(* CODESYS project hmi_library.library
   Author: AMKO-Engineering
   Placeholder: HMI_Library
   Title: HMI_Library
   Version: 1.0.0.3
   Description: Basic HMI screens for use with Utilities and device libraries
   Company: AMKO-Engineering

Project tree, tasks and I/O mapping:
  libraries: CmpBitmapPool, 3.5.7.0 (System); Device_Library, 1.2.0.3 (AMKO-Engineering); System_Library, * (AMKO-Engineering); Utilities_Library, 1.2.0.3 (AMKO-Engineering); VisuDialogs, 3.5.12.0 (System)
  BaseScreens/
  GVL/
    data type E_StartVisu
    global variables GVL_HMI
  IconsAndPictures/
    Backgrounds/
      Background.svg
      Background_Bottom.svg
      Background_Bottomzonder knop.png
      Background_Sides.svg
      image pool BackgroundImagePool
      Emergency Stop Active.jpg
    Buttons/
      Home Button/
        Home Settings switch.png
        Home_Settings switch.svg
        Home-Settings Switch Pushed.png
        Home-Settings Switch Pushed.svg
      Screen Buttons/
        Power Off Pressed.png
        Power off.png
        To Parameter Screen Pressed.png
        To Parameter Screen Pressed.svg
        To Parameter Screen.png
        To Parameter Screen.svg
      image pool ButtonImagePool
    Logos/
      Amko Basis.svg
      Logo Dark blue.svg
      image pool LogoPool
  00000000-0000-0000-0000-000000000000|IconsAndPictures\Backgrounds\Background.svg
  00000000-0000-0000-0000-000000000000|IconsAndPictures\Backgrounds\Background_Bottom.svg
  00000000-0000-0000-0000-000000000000|IconsAndPictures\Backgrounds\Background_Bottomzonder knop.png
  00000000-0000-0000-0000-000000000000|IconsAndPictures\Backgrounds\Background_Sides.svg
  00000000-0000-0000-0000-000000000000|IconsAndPictures\Backgrounds\Emergency Stop Active.jpg
  00000000-0000-0000-0000-000000000000|IconsAndPictures\Buttons\Home Button\Home Settings switch.png
  00000000-0000-0000-0000-000000000000|IconsAndPictures\Buttons\Home Button\Home_Settings switch.svg
  00000000-0000-0000-0000-000000000000|IconsAndPictures\Buttons\Home Button\Home-Settings Switch Pushed.png
  00000000-0000-0000-0000-000000000000|IconsAndPictures\Buttons\Home Button\Home-Settings Switch Pushed.svg
  00000000-0000-0000-0000-000000000000|IconsAndPictures\Buttons\Screen Buttons\Power Off Pressed.png
  00000000-0000-0000-0000-000000000000|IconsAndPictures\Buttons\Screen Buttons\Power off.png
  00000000-0000-0000-0000-000000000000|IconsAndPictures\Buttons\Screen Buttons\To Parameter Screen Pressed.png
  00000000-0000-0000-0000-000000000000|IconsAndPictures\Buttons\Screen Buttons\To Parameter Screen Pressed.svg
  00000000-0000-0000-0000-000000000000|IconsAndPictures\Buttons\Screen Buttons\To Parameter Screen.png
  00000000-0000-0000-0000-000000000000|IconsAndPictures\Buttons\Screen Buttons\To Parameter Screen.svg
  00000000-0000-0000-0000-000000000000|IconsAndPictures\Logos\Amko Basis.svg
  00000000-0000-0000-0000-000000000000|IconsAndPictures\Logos\Logo Dark blue.svg
  InputFunctions/
    function block FB_HMIInputBase [ST]: SetHMIInstructions, SetOutputToPLC
    function block FB_HMILREALInput [ST]: SetOutputToPLC
  Screens/
    Backgrounds/
      visualisation BackgroundNoButton
    EventsAndMessage/
      visualisation BasicMessageScreen
      visualisation EstopScreen
    Manual/
      DeviceScreens/
        visualisation VisuAnalogOutControl
        visualisation VisuAnlogInputControl
        visualisation VisuAxisControl
        visualisation VisuCylinderControl
        visualisation VisuDigitalInputControl
        visualisation VisuDigitalOutControl
        visualisation VisuPushbuttonLightControl
        visualisation VisuPWMControl
        visualisation VisuUndefinedControl
        visualisation VisuValveControl
      visualisation ManualControl
    Parameter/
      visualisation ParameterScreen
    Startup Screen/
      visualisation LogoScreen
      visualisation StartScreen
  TextLists/
    text list E_ComponentTypes
    text list E_FaultTypes
    text list E_Locations
    text list E_MessageNumbers
    text list E_ParameterNames
    text list GlobalTextList
    text list TL_MessageDiscriptions
*)

// GVL/E_StartVisu
{attribute 'qualified_only'}
{attribute 'strict'}
TYPE E_StartVisu :
(
	Logo := 0,
	Parameter,
	Manual
);
END_TYPE

// GVL/GVL_HMI
{attribute 'qualified_only'}
VAR_GLOBAL
	nStartVisu	: E_StartVisu := E_StartVisu.Logo ;
END_VAR

// InputFunctions/FB_HMIInputBase
FUNCTION_BLOCK ABSTRACT FB_HMIInputBase //Base function for HMI inputs
VAR_INPUT
	bEnable : BOOL := TRUE ;
END_VAR
VAR_OUTPUT
	bInVisible			: BOOL := TRUE ; // input is visible (standard := NOT bEnable )
	bDeactivateInput	: BOOL := TRUE ; // input is enabled (Standard := bEnable)
END_VAR
VAR
END_VAR

SetHMIInstructions();

METHOD INTERNAL SetHMIInstructions : BOOL
VAR_INPUT
END_VAR
bInVisible 			:= NOT bEnable ;
bDeactivateInput	:= NOT bEnable ;
END_METHOD

METHOD ABSTRACT SetOutputToPLC : BOOL
VAR_INPUT
END_VAR
END_METHOD

END_FUNCTION_BLOCK

// InputFunctions/FB_HMILREALInput
FUNCTION_BLOCK PUBLIC FB_HMILREALInput EXTENDS FB_HMIInputBase // Analog value input from HMI
VAR_INPUT
	fInputFromHMI	: LREAL ;
END_VAR
VAR_OUTPUT
	fOutputToPLC	: LREAL ;
END_VAR
VAR
END_VAR

// call base function 
SUPER^();

// Set output to PLC
SetOutputToPLC();

METHOD PUBLIC SetOutputToPLC : BOOL
VAR_INPUT
END_VAR
IF bEnable THEN 
	fOutputToPLC := fInputFromHMI ;
END_IF
END_METHOD

END_FUNCTION_BLOCK

// Screens/Backgrounds/BackgroundNoButton
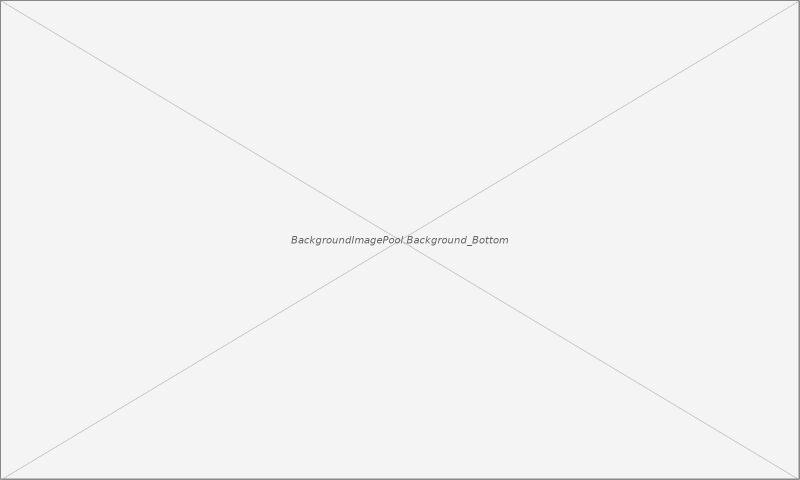
VISUALIZATION BackgroundNoButton  // 800x480
    Image (0,0 800x480), invisible if: SystemBase.bSystemOK, input disabled if: SystemBase.bSystemOK, image: BackgroundImagePool.Emergency Stop Active
    Image (0,0 800x480), image: BackgroundImagePool.Background_Bottom
END_VISUALIZATION

// Screens/EventsAndMessage/BasicMessageScreen
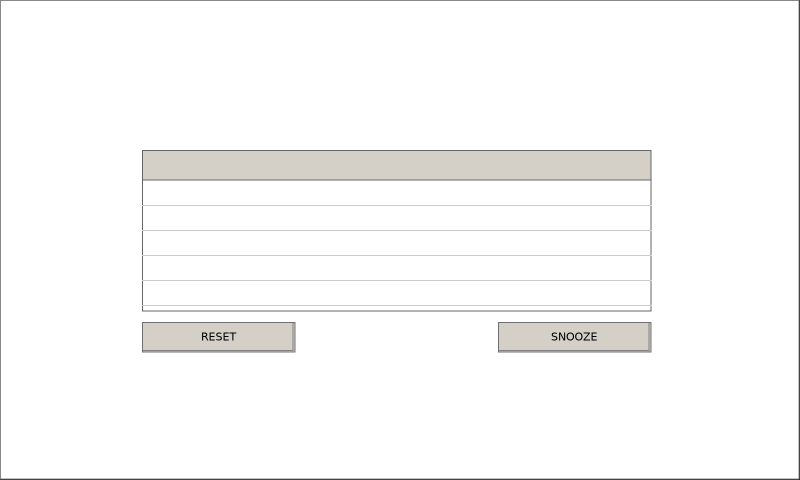
VISUALIZATION BasicMessageScreen  // 800x480
    Rectangle (0,0 800x480)
    Table (142,150 509x161), data array: Utilities_Library.GVL_Message.arActiveFaults
        p3854506369: Utilities_Library.GVL_Message.arActiveFaults[INDEX].Active
        p1892666644: Utilities_Library.GVL_Message.arActiveFaults[INDEX].FaultType
        p338671338: Utilities_Library.GVL_Message.arActiveFaults[INDEX].MessageNumber
        p2170511999: Utilities_Library.GVL_Message.arActiveFaults[INDEX].LocationNumber
        p3723444502: Utilities_Library.GVL_Message.arActiveFaults[INDEX].Discription
        p1218418051: Utilities_Library.GVL_Message.arActiveFaults[INDEX].LocationName
        p746581629: Utilities_Library.GVL_Message.arActiveFaults[INDEX].ComponentType
        p3104783080: Utilities_Library.GVL_Message.arActiveFaults[INDEX].StartTime
        p2501879983: Utilities_Library.GVL_Message.arActiveFaults[INDEX].EndTime
        p7306298: Utilities_Library.GVL_Message.arActiveFaults[INDEX].nModuleID
        p1933151965: Utilities_Library.GVL_Message.arActiveFaults[INDEX].FullFaultId
    Button (142,322 153x30), "RESET"
        tap Utilities_Library.GVL_Message.bResetFaults
    Button (498,322 153x30), "SNOOZE"
        tap Utilities_Library.GVL_Message.bCmdSnoozeMessage
END_VISUALIZATION

// Screens/EventsAndMessage/EstopScreen
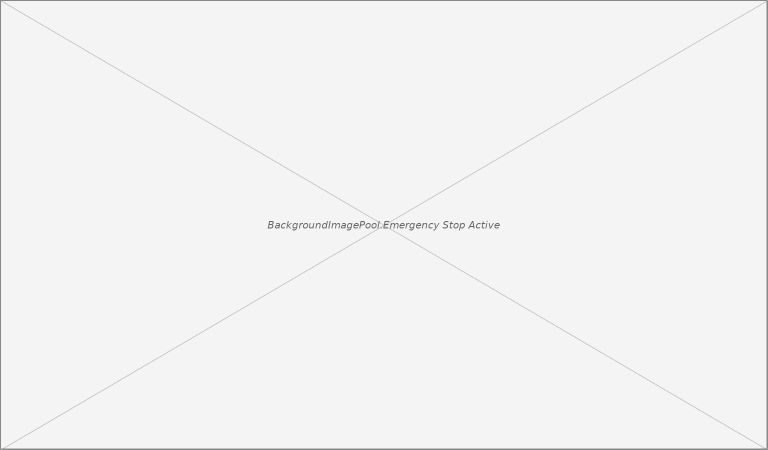
VISUALIZATION EstopScreen  // 768x450
    Image (0,0 768x450), image: BackgroundImagePool.Emergency Stop Active
END_VISUALIZATION

// Screens/Manual/DeviceScreens/VisuAnalogOutControl
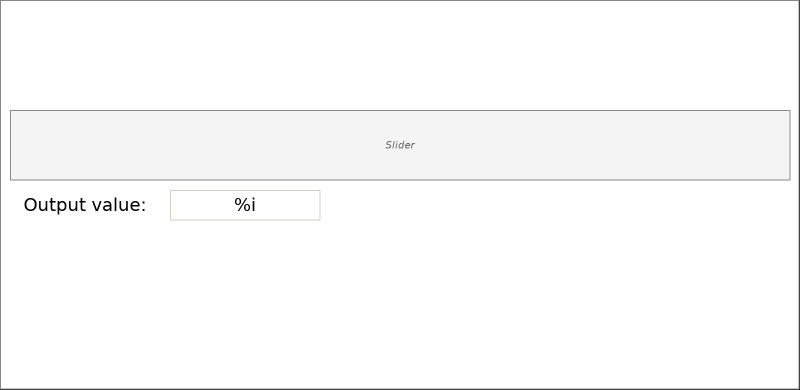
VISUALIZATION VisuAnalogOutControl  // 800x390
    Rectangle (0,0 800x390)
    Slider (10,110 780x70), variable: GVL_DevManual.fbManualControler.pDevAnalogOut^.fCmdValue, scale 0..100
    Textfield (170,190 150x30), "%i", text variable: GVL_DevManual.fbManualControler.pDevAnalogOut^.fCmdValue
        OnMouseClick: write the text variable via VisuDialogs.Numpad
    Label (10,190 150x30), "Output value:"
END_VISUALIZATION

// Screens/Manual/DeviceScreens/VisuAnlogInputControl
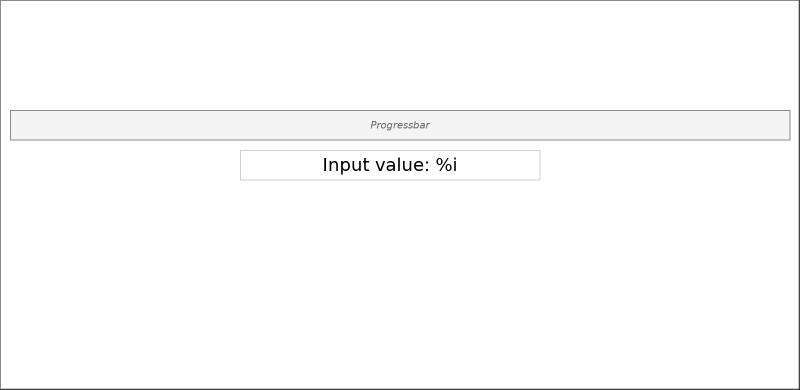
VISUALIZATION VisuAnlogInputControl  // 800x390
    Rectangle (0,0 800x390)
    Progressbar (10,110 780x30), variable: GVL_DevManual.fbManualControler.pDevAnalogInput^.fValue
    Textfield (240,150 300x30), "Input value: %i", text variable: GVL_DevManual.fbManualControler.pDevAnalogInput^.fValue
END_VISUALIZATION

// Screens/Manual/DeviceScreens/VisuAxisControl
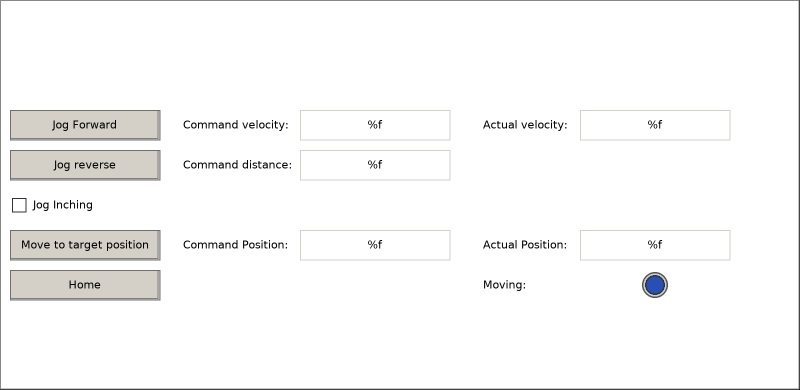
VISUALIZATION VisuAxisControl  // 800x390
    Rectangle (0,0 800x390)
    Button (10,110 150x30), "Jog Forward"
        tap GVL_DevManual.fbManualControler.pDevAxis^.stManualCtrl.bCmdJogForward
    Button (10,150 150x30), "Jog reverse"
        tap GVL_DevManual.fbManualControler.pDevAxis^.stManualCtrl.bCmdJogReverse
    Button (10,230 150x30), "Move to target position"
        tap GVL_DevManual.fbManualControler.pDevAxis^.stManualCtrl.bCmdToPos
    Button (10,270 150x30), "Home"
        tap GVL_DevManual.fbManualControler.pDevAxis^.stManualCtrl.bCmdHome
    Checkbox (10,190 150x30), "Jog Inching", variable: GVL_DevManual.fbManualControler.pDevAxis^.stManualCtrl.bCmdInching
    Label (180,150 120x30), "Command distance:"
    Label (180,110 120x30), "Command velocity:"
    Label (180,230 120x30), "Command Position:"
    Textfield (300,110 150x30), "%f", text variable: GVL_DevManual.fbManualControler.pDevAxis^.stManualCtrl.fVelocity
        OnMouseDown: write the text variable via VisuDialogs.Numpad
    Textfield (300,150 150x30), "%f", text variable: GVL_DevManual.fbManualControler.pDevAxis^.stManualCtrl.fDistance
        OnMouseDown: write the text variable via VisuDialogs.Numpad
    Textfield (300,230 150x30), "%f", text variable: GVL_DevManual.fbManualControler.pDevAxis^.stManualCtrl.fPosition
        OnMouseDown: write the text variable via VisuDialogs.Numpad
    Label (480,110 100x30), "Actual velocity:"
    Label (480,230 100x30), "Actual Position:"
    Textfield (580,230 150x30), "%f", text variable: GVL_DevManual.fbManualControler.pDevAxis^.fActPosition
        OnMouseDown: write the text variable via VisuDialogs.Numpad
    Textfield (580,110 150x30), "%f", text variable: GVL_DevManual.fbManualControler.pDevAxis^.fVelocity
        OnMouseDown: write the text variable via VisuDialogs.Numpad
    Lamp1 (580,270 150x30), variable: GVL_DevManual.fbManualControler.pDevAxis^.AxisRef.Status.Moving, style: Lamp-Lamp1-Blue
    Label (480,270 100x30), "Moving:"
END_VISUALIZATION

// Screens/Manual/DeviceScreens/VisuCylinderControl
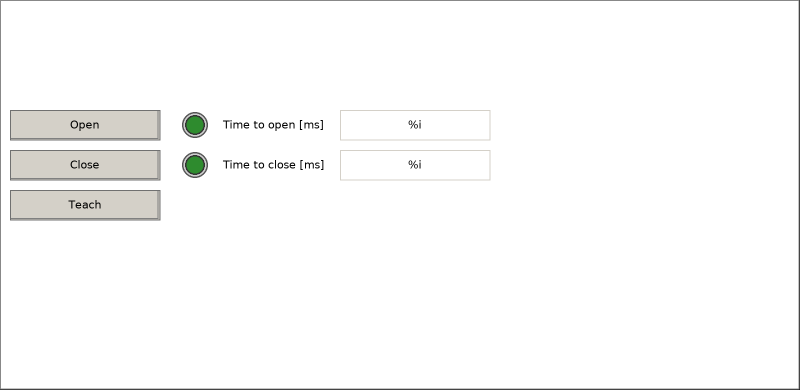
VISUALIZATION VisuCylinderControl  // 800x390
    Rectangle (0,0 800x390)
    Button (10,110 150x30), "Open"
        tap GVL_DevManual.fbManualControler.pDevCylinder^.stManualCtrl.bCmdOpen
    Button (10,150 150x30), "Close"
        tap GVL_DevManual.fbManualControler.pDevCylinder^.stManualCtrl.bCmdClose
    Lamp1 (180,110 30x30), variable: GVL_DevManual.fbManualControler.pDevCylinder^.bFco_Open, style: Lamp-Lamp1-Green
    Button (10,190 150x30), "Teach"
        toggle GVL_DevManual.fbManualControler.pDevCylinder^.stManualCtrl.bCmdTeach
    Lamp1 (180,150 30x30), variable: GVL_DevManual.fbManualControler.pDevCylinder^.bFco_Closed, style: Lamp-Lamp1-Green
    Label (220,110 100x30), "Time to open [ms]"
    Label (220,150 100x30), "Time to close [ms]"
    Textfield (340,150 150x30), "%i", text variable: GVL_DevManual.fbManualControler.pDevCylinder^.stParTimeToClose.fValue
        OnMouseClick: write the text variable via VisuDialogs.Numpad, min 0
    Textfield (340,110 150x30), "%i", text variable: GVL_DevManual.fbManualControler.pDevCylinder^.stParTimeToOpen.fValue
        OnMouseClick: write the text variable via VisuDialogs.Numpad, min 0
END_VISUALIZATION

// Screens/Manual/DeviceScreens/VisuDigitalInputControl
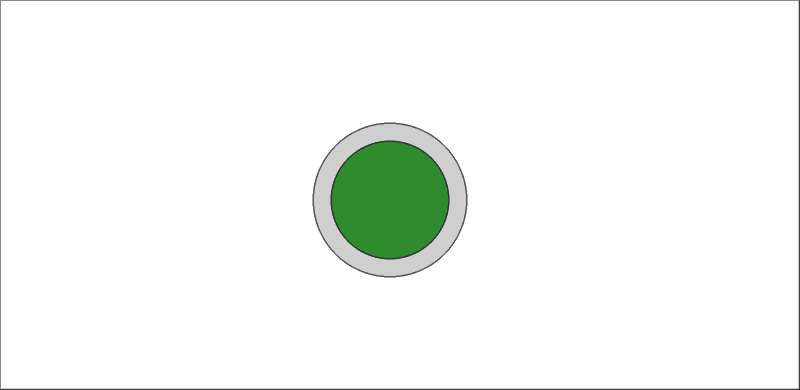
VISUALIZATION VisuDigitalInputControl  // 800x390
    Rectangle (0,0 800x390)
    Lamp1 (300,110 180x180), variable: GVL_DevManual.fbManualControler.pDevDigitalInput^.bFcoInputActive, style: Lamp-Lamp1-Green
END_VISUALIZATION

// Screens/Manual/DeviceScreens/VisuDigitalOutControl
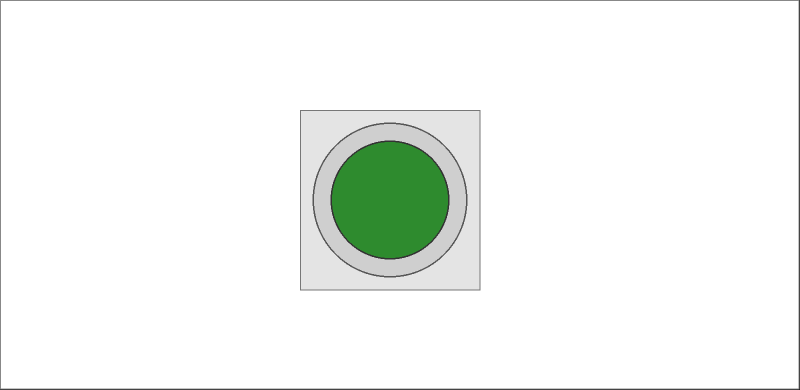
VISUALIZATION VisuDigitalOutControl  // 800x390
    Rectangle (0,0 800x390)
    PushSwitch (300,110 180x180), variable: GVL_DevManual.fbManualControler.pDevDigitalOut^.bCmdOn, behaviour: TOGGLE, style: Switch-PushSwitch-Green
END_VISUALIZATION

// Screens/Manual/DeviceScreens/VisuPushbuttonLightControl
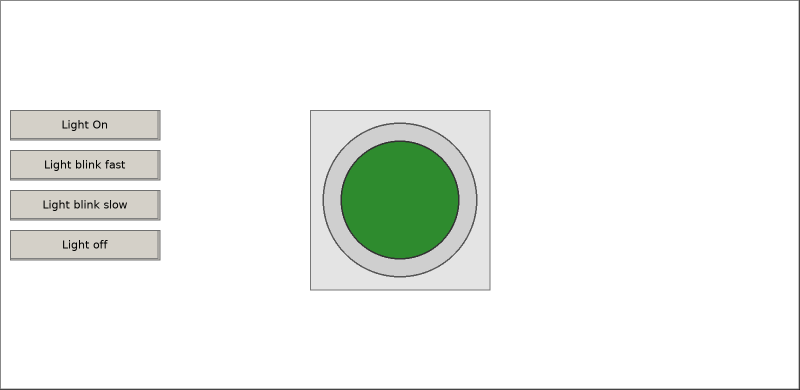
VISUALIZATION VisuPushbuttonLightControl  // 800x390
    Rectangle (0,0 800x390)
    PushSwitch (310,110 180x180), variable: GVL_DevManual.fbManualControler.pDevPBL^.bFcoInputActive, behaviour: TOGGLE, style: Switch-PushSwitch-Green
    Button (10,110 150x30), "Light On"
        tap GVL_DevManual.fbManualControler.pDevPBL^.fbLight.bCmdOn
    Button (10,150 150x30), "Light blink fast"
        tap GVL_DevManual.fbManualControler.pDevPBL^.fbLight.bCmdBlinkFast
    Button (10,190 150x30), "Light blink slow"
        tap GVL_DevManual.fbManualControler.pDevPBL^.fbLight.bCmdBlinkSlow
    Button (10,230 150x30), "Light off"
        tap GVL_DevManual.fbManualControler.pDevPBL^.fbLight.bCmdOff
END_VISUALIZATION

// Screens/Manual/DeviceScreens/VisuPWMControl
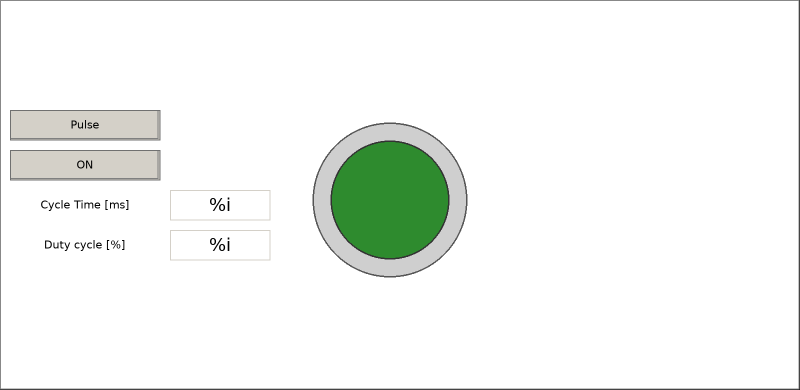
VISUALIZATION VisuPWMControl  // 800x390
    Rectangle (0,0 800x390)
    Lamp1 (300,110 180x180), variable: GVL_DevManual.fbManualControler.pDevPWMController^.qbOutput, style: Lamp-Lamp1-Green
    Button (10,110 150x30), "Pulse"
        toggle GVL_DevManual.fbManualControler.pDevPWMController^.bCmdPWMCycle
    Button (10,150 150x30), "ON"
        tap GVL_DevManual.fbManualControler.pDevPWMController^.bCmdOn
    Textfield (170,190 100x30), "%i", text variable: GVL_DevManual.fbManualControler.pDevPWMController^.nPeriodLength
        OnMouseUp: write the text variable via VisuDialogs.Numpad
    Label (10,190 150x30), "Cycle Time [ms]"
    Label (10,230 150x30), "Duty cycle [%]"
    Textfield (170,230 100x30), "%i", text variable: GVL_DevManual.fbManualControler.pDevPWMController^.nDutyCycle
        OnMouseClick: write the text variable via VisuDialogs.Numpad, min 0, max 100
END_VISUALIZATION

// Screens/Manual/DeviceScreens/VisuUndefinedControl
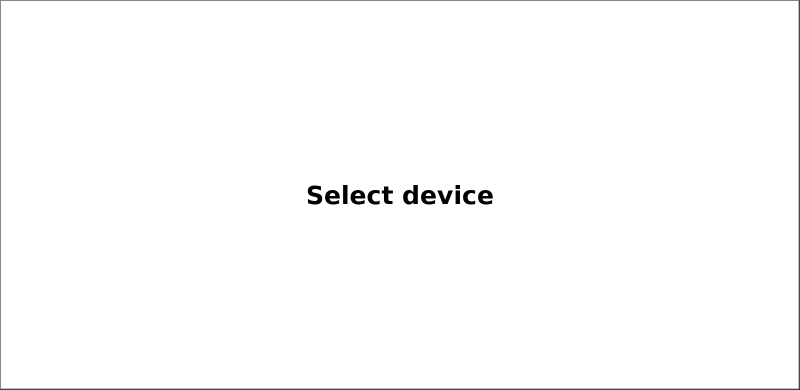
VISUALIZATION VisuUndefinedControl  // 800x390
    Rectangle (0,0 800x390)
    Label (0,0 800x390), "Select device"
END_VISUALIZATION

// Screens/Manual/DeviceScreens/VisuValveControl
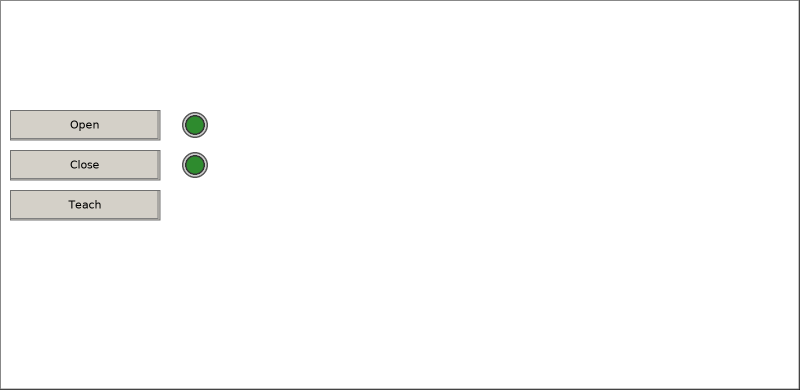
VISUALIZATION VisuValveControl  // 800x390
    Rectangle (0,0 800x390)
    Button (10,110 150x30), "Open"
        tap GVL_DevManual.fbManualControler.pDevValve^.stManualCtrl.bCmdOpen
    Button (10,150 150x30), "Close"
        tap GVL_DevManual.fbManualControler.pDevValve^.stManualCtrl.bCmdClose
    Lamp1 (180,110 30x30), variable: GVL_DevManual.fbManualControler.pDevValve^.bFco_Open, style: Lamp-Lamp1-Green
    Button (10,190 150x30), "Teach"
        toggle GVL_DevManual.fbManualControler.pDevValve^.stManualCtrl.bCmdTeach
    Lamp1 (180,150 30x30), variable: GVL_DevManual.fbManualControler.pDevValve^.bFco_Closed, style: Lamp-Lamp1-Green
END_VISUALIZATION

// Screens/Manual/ManualControl
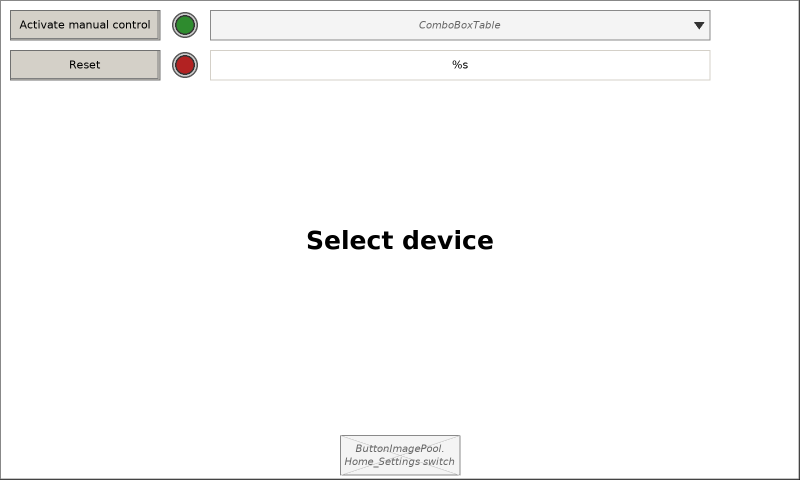
VISUALIZATION ManualControl  // 800x480
    Frame (0,0 800x480), input disabled if: GVL_DevManual.fbManualControler.bDisableManualInputs, frame switch variable: GVL_DevManual.fbManualControler.eDevType
        shows VisuUndefinedControl()
        shows VisuValveControl()
        shows VisuCylinderControl()
        shows VisuAxisControl()
        shows VisuPushbuttonLightControl()
        shows VisuDigitalInputControl()
        shows VisuAnlogInputControl()
        shows VisuDigitalOutControl()
        shows VisuAnalogOutControl()
        shows VisuPWMControl()
    Button (10,10 150x30), "Activate manual control", pressed state: GVL_DevManual.fbManualControler.bManualActive
        toggle GVL_DevManual.fbManualControler.bManualActive
    Lamp1 (170,50 30x30), tooltip "component fault active", variable: GVL_DevManual.fbManualControler.bErroractive, style: Lamp-Lamp1-Red
    Lamp1 (170,10 30x30), tooltip "Manual control active", variable: GVL_DevManual.fbManualControler.bManual, style: Lamp-Lamp1-Green
    Textfield (210,50 500x30), "%s", text variable: GVL_DevManual.fbManualControler.sDeviceState
    Button (10,50 150x30), "Reset"
        tap GVL_DevManual.fbManualControler.bReset
    ComboBoxTable (210,10 500x30), variable: GVL_DevManual.fbManualControler.nCmdLookupindex, data array: GVL_DevManual.fbManualControler.arDeviceArray
        p3854506369: GVL_DevManual.fbManualControler.arDeviceArray[INDEX].sName
        p1892666644: GVL_DevManual.fbManualControler.arDeviceArray[INDEX].sType
        p338671338: GVL_DevManual.fbManualControler.arDeviceArray[INDEX].pFunction^
        p1128707560: GVL_DevManual.fbManualControler.nNumberOfDevices
    Image (340,435 120x40), image: ButtonImagePool.Home_Settings switch
        OnMouseClick: execute { GVL_HMI.nStartVisu := E_StartVisu.Logo ; }
        OnMouseClick:  ToggleVariable=GVL_Parameters.fbParameterHandler.bCmdParFileWrite
END_VISUALIZATION

// Screens/Parameter/ParameterScreen
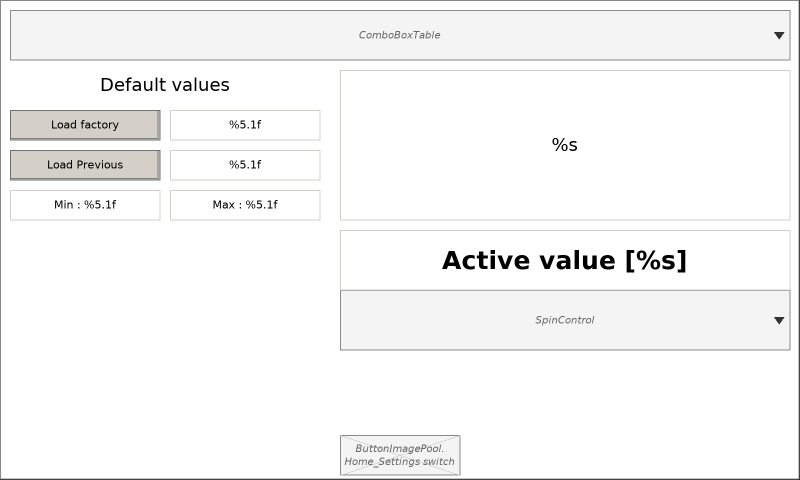
VISUALIZATION ParameterScreen  // 800x480
    Rectangle (0,0 800x480)
    ComboBoxTable (10,10 780x50), variable: GVL_Parameters.fbParameterHandler.nLookupIndex, data array: GVL_Parameters.fbParameterHandler.arParameters
        p1128707560: GVL_Parameters.fbParameterHandler.nNumberOfParameters
        p3854506369: GVL_Parameters.fbParameterHandler.arParameters[INDEX].nNumber
        p1892666644: GVL_Parameters.fbParameterHandler.arParameters[INDEX].sName
        p338671338: GVL_Parameters.fbParameterHandler.arParameters[INDEX].sType
        p2170511999: GVL_Parameters.fbParameterHandler.arParameters[INDEX].pParameter^
    Group (10,70 310x150)
        Button (0,40 150x30), "Load factory"
            tap GVL_Parameters.fbParameterHandler.bCmdLoadfactory
        Label (0,0 310x30), "Default values"
        Textfield (160,40 150x30), "%5.1f", text variable: GVL_Parameters.fbParameterHandler.arParameters[GVL_Parameters.fbParameterHandler.nLookupIndex].pParameter^.fFactory
            OnMouseClick: write the text variable via VisuDialogs.Numpad, min GVL_Parameters.fbParameterHandler.arParameters[GVL_Parameters.fbParameterHandler.nLookupIndex].pParameter^.fMinimum, max GVL_Parameters.fbParameterHandler.arParameters[GVL_Parameters.fbParameterHandler.nLookupIndex].pParameter^.fMaximum
        Button (0,80 150x30), "Load Previous"
            tap GVL_Parameters.fbParameterHandler.bCmdLoadFromPrevious
        Textfield (160,80 150x30), "%5.1f", text variable: GVL_Parameters.fbParameterHandler.arParameters[GVL_Parameters.fbParameterHandler.nLookupIndex].pParameter^.fSaved
        Textfield (160,120 150x30), "Max : %5.1f", text variable: GVL_Parameters.fbParameterHandler.arParameters[GVL_Parameters.fbParameterHandler.nLookupIndex].pParameter^.fMaximum
            OnMouseClick: write the text variable via VisuDialogs.Numpad
        Textfield (0,120 150x30), "Min : %5.1f", text variable: GVL_Parameters.fbParameterHandler.arParameters[GVL_Parameters.fbParameterHandler.nLookupIndex].pParameter^.fMinimum
            OnMouseClick: write the text variable via VisuDialogs.Numpad
    Textfield (340,70 450x150), "%s", text variable: GVL_Parameters.fbParameterHandler.arParameters[GVL_Parameters.fbParameterHandler.nLookupIndex].pParameter^.sDiscription
    SpinControl (340,290 450x60), variable: GVL_Parameters.fbParameterHandler.arParameters[GVL_Parameters.fbParameterHandler.nLookupIndex].pParameter^.fValue
        p576042468: GVL_Parameters.fbParameterHandler.arParameters[GVL_Parameters.fbParameterHandler.nLookupIndex].pParameter^.fMinimum
        p651134158: GVL_Parameters.fbParameterHandler.arParameters[GVL_Parameters.fbParameterHandler.nLookupIndex].pParameter^.fMaximum
        OnMouseClick: write the text variable via VisuDialogs.Numpad, min GVL_Parameters.fbParameterHandler.arParameters[GVL_Parameters.fbParameterHandler.nLookupIndex].pParameter^.fMinimum, max GVL_Parameters.fbParameterHandler.arParameters[GVL_Parameters.fbParameterHandler.nLookupIndex].pParameter^.fMaximum
    Textfield (340,230 450x60), "Active value [%s]", text variable: GVL_Parameters.fbParameterHandler.arParameters[GVL_Parameters.fbParameterHandler.nLookupIndex].pParameter^.sUnit
    Image (340,435 120x40), image: ButtonImagePool.Home_Settings switch
        OnMouseClick: execute { GVL_HMI.nStartVisu := E_StartVisu.Logo ; }
        OnMouseClick:  ToggleVariable=GVL_Parameters.fbParameterHandler.bCmdParFileWrite
END_VISUALIZATION

// Screens/Startup Screen/LogoScreen
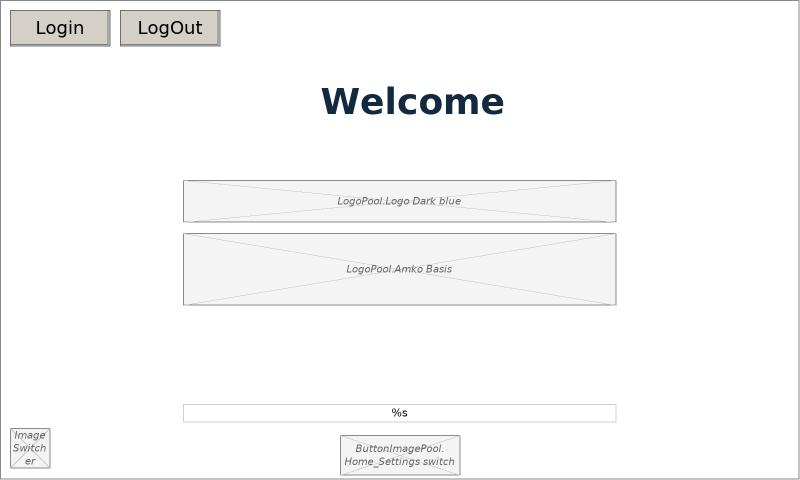
VISUALIZATION LogoScreen  // 800x480
    Rectangle (0,0 800x480)
    Textfield (258,76 310x51), "Welcome"
    Image (183,180 433x42), image: LogoPool.Logo Dark blue
    Image (183,233 433x72), image: LogoPool.Amko Basis
    InvisibleInput (728,10 62x60)
        OnMouseClick: execute { GVL_HMI.nStartVisu := E_StartVisu.Manual; }
    Button (10,10 100x36), "Login"
        OnMouseClick:  Type=Login
    Textfield (183,404 433x18), "%s", tooltip "Operator messagages", text variable: GVL_Message.sOPeratorMessage
    Button (120,10 100x36), "LogOut"
        OnMouseClick:  Type=Logout
    ImageSwitcher (10,428 40x40), variable: SystemBase.fbCmdPowerOff.Istatus, background image: ButtonImagePool.Power Off Pressed, image: ButtonImagePool.Power off, behaviour: TAP
    Image (340,435 120x40), image: ButtonImagePool.Home_Settings switch
        OnMouseClick: execute { GVL_HMI.nStartVisu := E_StartVisu.Parameter; }
END_VISUALIZATION

// Screens/Startup Screen/StartScreen
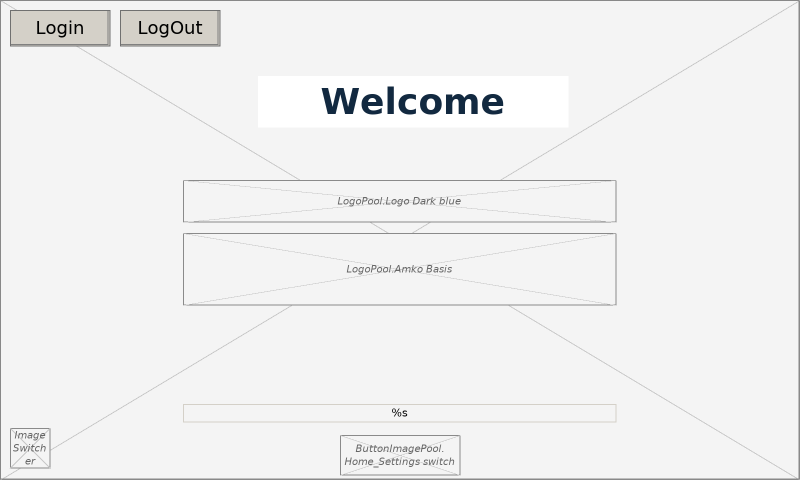
VISUALIZATION StartScreen  // 800x480
    Frame (0,0 800x480)
        shows BackgroundNoButton()
    Frame (0,0 800x480), frame switch variable: GVL_HMI.nStartVisu
        shows LogoScreen()
        shows ParameterScreen()
        shows ManualControl()
END_VISUALIZATION

(* text list E_ComponentTypes (id | default)
  0 | NA
  10 | Cylinder
  11 | Axis
  20 | EstopButton
  21 | EstopBumper
  22 | Pushbutton
  23 | Switch
  30 | SafeIO
  31 | Rio_Box
  32 | Rio_Slot
  33 | Encoder
  34 | DiSensor
  40 | ServoDrive
  50 | HMI
  51 | RemoteOS
  52 | RemoteDB
  60 | Assembly
  61 | SubAssembly
  100 | MainProgram
  101 | StepProgram
  102 | FunctionBlock
   |  *)

(* text list E_FaultTypes (id | default)
  0 | NA
  1 | OM
  2 | MC
  3 | CF
  4 | FF
   |  *)

(* text list E_Locations (id | default)
  0 | Main PLC
  1 | 230V Main supply
  2 | 24V Main supply
  3 | Main air supply
  4 | Main Screen
  5 | Main IO
   |  *)

(* text list E_MessageNumbers (id | default)
  0 | NA_NoMessage
  1 | FF_Unknown
  2 | FF_NoCommunication
  3 | FF_ComunicationFault
  4 | FF_Overload
  5 | FF_EncoderFault
  6 | FF_SlaveFault
  7 | FF_AxisFault
  8 | FF_DriveFault
  9 | FF_Collision
  100 | CF_FeedbackFault
  101 | CF_WrongDirection
  102 | CF_MoveToFast
  103 | CF_MoveToSlow
  104 | CF_WrongPosition
  105 | CF_Obstruction
  200 | MC_WaitingForproduct
  201 | MC_WaitingForOperator
  202 | MC_WaitingForModule
  203 | MC_WaitingForMaster
  204 | MC_WaitingForSlave
  205 | MC_WrongPosition
  300 | OM_AlmostEmpty
  301 | OM_Finished
  302 | OM_ready
  900 | FF_MessageTest
  901 | CF_MessageTest
  902 | MC_MessageTest
  903 | OM_MessageTest
   |  *)

(* text list E_ParameterNames (id | default)
  0 | Mpar_StitchLengthLong
  1 | MPar_StitchLengthShort
  2 | MPar_MaxSpeed
  3 | Mpar_MinSpeed
  4 | Mpar_ManualMaxSpeed
  5 | Mpar_BacktackSpeed
  6 | Mpar_SlowEndSpeed
  7 | Mpar_HomingSpeed
  8 | Mpar_CuttingSpeed
  9 | Mpar_MaxAcceleration
  10 | Mpar_MaxDeceleration
  11 | Mpar_Jerk
  12 | Mpar_BacktackAcceleration
  13 | Mpar_BacktackDeceleration
  14 | Mpar_TransferAcceleration
  15 | Mpar_TransferDeceleration
  16 | Mpar_CylinderTimeoutMargin
  17 | Cpar_NeedleSensorPos
  18 | Cpar_NeedlePosUp
  19 | Cpar_NeedlePosInMaterial
  20 | Cpar_NeedleposDown
  21 | Cpar_NeedlePosStartCut
  22 | Cpar_NeedlePosStopCut
  23 | Cpar_NeedlePosEndCut
  24 | Cpar_NeedlePosRelTensCut
  25 | Cpar_NeedlePosHoldThread
  26 | Cpar_NeedlePosStartRelTension
  27 | Cpar_NeedlePosStopRelTension
  28 | Cpar_NeedlePosChangeDirUp
  29 | Cpar_NeedlePosClearStart
  30 | Cpar_NeedlePosClearEnd
  31 | Cpar_NeedlePosRef
  32 | Cpar_NeedlePosPause
  33 | Cpar_SensorPreEdgeDetDistance
  34 | Cpar_sensorEdgeDetDistance
  35 | Opar_NeedleSensorPos
  36 | Opar_NeedlePosUp
  37 | Opar_NeedlePosInMaterial
  38 | Opar_NeedleposDown
  39 | Opar_NeedlePosStartCut
  40 | Opar_NeedlePosStopCut
  41 | Opar_NeedlePosEndCut
  42 | Opar_NeedlePosRelTensCut
  43 | Opar_NeedlePosHoldThread
  44 | Opar_NeedlePosStartRelTension
  45 | Opar_NeedlePosStopRelTension
  46 | Opar_NeedlePosChangeDir
  47 | Opar_NeedlePosClearStart
  48 | Opar_NeedlePosClearEnd
  49 | Opar_NeedlePosPause
  50 | Ppar_BacktackStitchStartFwd
  51 | Ppar_BacktackStitchStartRev
  52 | Ppar_BacktackStitchEndFwd
  53 | Ppar_BacktackStitchEndRev
  54 | Ppar_AutomaticSpeed
  55 | Ppar_StitchStretch
  56 | Ppar_ThreadLengthAdition
  57 | Ppar_ThreadBreakDelay
  58 | Mpar_MaxVelocity
  59 | Mpar_MinVelocity
  60 | Mpar_ManualMaxVelocity
  61 | Mpar_MLTMaxAcceleration
  62 | Mpar_MLTMaxDeceleration
  63 | Mpar_TraverseLength
  64 | Mpar_CylTimeOutMargine
  65 | Mpar_HomingVelocity
  66 | Mpar_SewingcartLength
  67 | Mpar_ClampCartLength
  68 | Mpar_MaxClampCartVelocity
  69 | Mpar_TraverseReturnVelocity
  70 | Mpar_ToStartvelocity
  71 | Mpar_InspectionDistance
  72 | Cpar_PosHoming
  73 | Cpar_PosSuportCyl_1
  74 | Cpar_PosSuportCyl_2
  75 | Cpar_PosSuportCyl_3
  76 | Cpar_PosService
  77 | Cpar_PosBobinChange
  78 | Cpar_PosEnd
  79 | Cpar_TimeBaseClampsClose
  80 | Cpar_TimeBaseClampsRel
  81 | Cpar_TimeCartClampsClose
  82 | Cpar_TimeCartClampsRel
  83 | Cpar_TimeCartBrakeApply
  84 | Cpar_TimeCartBrakeRel
  85 | Cpar_TimeSupportExp_1
  86 | Cpar_TimeSupportRet_1
  87 | Cpar_TimeSupportExp_2
  88 | Cpar_TimeSupportRet_2
  89 | Cpar_TimeSupportExp_3
  90 | Cpar_TimeSupportRet_3
  91 | Cpar_TimeBobinPlateClose
  92 | Cpar_TimeBobinPlateOpen
  93 | Cpar_PosFlagSewingcart
  94 | Cpar_PosSensorClampCart
  95 | Cpar_SupportCylWidth
  96 | Cpar_ClampCartFlagWidth
  97 | Cpar_PosMaterialStart
  98 | Opar_HomePosition
  99 | Opar_PosSuportCyl_1
  100 | Opar_PosSuportCyl_2
  101 | Opar_PosSuportCyl_3
  102 | Opar_PosService
  103 | Opar_PosBobinChange
  104 | Opar_PosEnd
  105 | Opar_PosMatStart
  106 | Ppar_ProductLenght
  107 | Ppar_ProductStretch
  108 | Ppar_StartStretchFactor
  109 | Ppar_StartStretchLength
  110 | Ppar_ReverseStretch
  111 | Ppar_MatBlowDistance
   |  *)

(* text list TL_MessageDiscriptions (id | default)
  0 | No message active
  1 | Unknown error occured
  2 | No communication detected
  3 | Communication error detected (does not match expected com)
  4 | Hardware overload detected
  5 | Encoder signal incorrect or not present
  6 | Slave system is has active fatal fault
  7 | Axis fault feedback
  8 | Axis drive fault
  9 | Collision detected between 2 or more parts of the machine
  100 | Hardware feedback is does not match expected
  101 | Hardware moving in incorrect direction
  102 | Hardware movement completion time is lower then minimum
  103 | Hardware movement maximum time was exceeded
  104 | Hardware is at different position then expected
  105 | Obstruction detected in movement path
  200 | Waiting for product
  201 | Waiting for operator action
  202 | Waiting for other module
  203 | Waiting Waiting for master
  204 | Waiting for slave
  205 | Action or command not possible in current position
  300 | Product is almost empty refif is required
  301 | Product or action is finished
  302 | Ready for new task
  900 | Fatal fault message test
  901 | Cycle fault message test
  902 | Missing condition message test
  903 | Operator message test
   |  *)
